(* IEC 61131-3 sources: Lasal/CPU_5344_V01/Class/cmMotor, 1 file *)

(* ---- cmMotor.st ---- *)
(*!
<Class
	Name               = "cmMotor"
	Revision           = "1.0"
	RealtimeTask       = "false"
	CyclicTask         = "true"
	DefCyclictime      = "10 ms"
	BackgroundTask     = "true"
	DefBackground      = "500 ms"
	Sigmatek           = "false"
	OSInterface        = "false"
	HighPriority       = "false"
	Automatic          = "false"
	UpdateMode         = "Prescan"
	SharedCommandTable = "true"
	Objectsize         = "(630,840)">
	<Channels>
		<Server Name="parMinTimeBetweenRev" Visualized="true" Initialize="false" WriteProtected="false" Retentive="File"/>
		<Server Name="parSpeed" Visualized="true" Initialize="false" WriteProtected="false" Retentive="false"/>
		<Server Name="parStartingTime" Visualized="true" Initialize="true" DefValue="2000" WriteProtected="false" Retentive="File"/>
		<Server Name="parTimeOutTime" Visualized="true" Initialize="true" DefValue="20000" WriteProtected="false" Retentive="File"/>
		<Server Name="stsBwd" Visualized="false" Initialize="false" WriteProtected="true" Retentive="false"/>
		<Server Name="stsFwd" Visualized="false" Initialize="false" WriteProtected="true" Retentive="false"/>
		<Server Name="stsStateRun" Visualized="true" Initialize="false" WriteProtected="false" Retentive="false"/>
		<Client Name="iFeedback" Required="false" Internal="false"/>
		<Client Name="iHWAlarm" Required="false" Internal="false" Comment="if used as btb, set sInvert"/>
		<Client Name="iThermFailure" Required="false" Internal="false" Comment="if used, connect thermical failure input,&#13;&#10;normally this input is high if there is a failure&#13;&#10;Else just set sInvert param"/>
		<Client Name="oBwd" Required="false" Internal="false"/>
		<Client Name="oFwd" Required="false" Internal="false"/>
		<Client Name="oSpeed" Required="false" Internal="false"/>
		<Client Name="sInvertFeedback" Required="false" Internal="false"/>
		<Client Name="sInvertHWAlarm" Required="false" Internal="false"/>
		<Client Name="sInvertThermFailure" Required="false" Internal="false"/>
		<Client Name="sMaxSpeedIn" Required="false" Internal="false" DefValue="1000"/>
		<Client Name="sMaxSpeedOut" Required="false" Internal="false" DefValue="10000"/>
		<Client Name="sMinSpeedIn" Required="false" Internal="false" DefValue="0"/>
		<Client Name="sMinSpeedOut" Required="false" Internal="false" DefValue="0"/>
	</Channels>
	<RevDoku>
		<Owner/>
		<Dokumentation Revision="0.1" Date="2019-12-13" Author="JdK&#13;&#10;" Company="vd" Description="calculation speed out is corrected, also added alarm for speed in out of borders"/>
	</RevDoku>
	<Network Name="cmMotor">
		<!-- List of Components in this network -->
		<Components>
			<Object
				Name       = "_base"
				Class      = "cmBase"
				Position   = "(218,120)"
				Visualized = "true">
				<Channels>
					<Server Name="ClassSvr"/>
					<Server Name="cmdHMI"/>
					<Server Name="ErrorNr"/>
					<Server Name="mode"/>
					<Server Name="state"/>
					<Server Name="stsHMI_RunsAllowed"/>
					<Server Name="stsInAlarm"/>
					<Server Name="stsIsInterlocked"/>
					<Client Name="id"/>
					<Client Name="nwEmOrUnit"/>
				</Channels>
			</Object>
		</Components>
		<Comments>
		</Comments>
		<!-- List of Connections in this network -->
		<Connections>
			<Connection Source="this.ClassSvr" Destination="_base.ClassSvr" Vertices="(1036,210),(864,210),"/>
			<Connection Source="this.state" Destination="_base.state" Vertices="(1036,270),(864,270),"/>
			<Connection Source="this.mode" Destination="_base.mode" Vertices="(1036,330),(864,330),"/>
			<Connection Source="this.cmdHMI" Destination="_base.cmdHMI" Vertices="(1036,390),(864,390),"/>
			<Connection Source="this.stsInAlarm" Destination="_base.stsInAlarm" Vertices="(1036,450),(864,510),"/>
			<Connection Source="this.stsIsInterlocked" Destination="_base.stsIsInterlocked" Vertices="(1036,510),(864,570),"/>
			<Connection Source="this.ErrorNr" Destination="_base.ErrorNr" Vertices="(1036,630),(864,690),"/>
			<Connection Source="_base.nwEmOrUnit" Destination="this.nwEmOrUnit" Vertices="(218,210),(38,210),"/>
			<Connection Source="_base.id" Destination="this.id" Vertices="(218,270),(38,270),"/>
			<Connection Source="this.stsHMI_RunsAllowed" Destination="_base.stsHMI_RunsAllowed" Vertices="(1036,570),(864,630),"/>
		</Connections>
		<!-- Headerfiles -->
		<Options>
		</Options>
	</Network>
</Class>
*)
#pragma using cmBase

cmMotor : CLASS
: cmBase
  //Servers:
	stsStateRun 	: SvrCh_motorPos;
	parTimeOutTime 	: SvrCh_UDINT;
	parStartingTime 	: SvrCh_UDINT;
	parMinTimeBetweenRev 	: SvrCh_UDINT;
	parSpeed 	: SvrCh_DINT;
	stsFwd 	: SvrCh_DINT;
	stsBwd 	: SvrCh_DINT;
  //Clients:
	iThermFailure 	: CltCh_DINT;
	iHWAlarm 	: CltCh_DINT;
	iFeedback 	: CltCh_DINT;
	oFwd 	: CltCh_DINT;
	oBwd 	: CltCh_DINT;
	oSpeed 	: CltCh_DINT;
	sInvertThermFailure 	: CltCh_DINT;
	sInvertHWAlarm 	: CltCh_DINT;
	sInvertFeedback 	: CltCh_DINT;
	sMinSpeedOut 	: CltCh_DINT;
	sMaxSpeedOut 	: CltCh_DINT;
	sMinSpeedIn 	: CltCh_DINT;
	sMaxSpeedIn 	: CltCh_DINT;
  //Variables:
		timerFeedback 	: strTimer;
		timerStarting 	: strTimer;
		timerFwdStopped 	: strTimer;
		timerBwdStopped 	: strTimer;
		feedbackConnected 	: DINT;
		tmpOSpeed 	: REAL;
		tmpThermFailure 	: DINT;
		tmpHWAlarm 	: DINT;
		tmpFeedback 	: DINT;
		tmpStartedHMI 	: DINT;
		tmpStartedCS 	: DINT;
		tmpOldSpeed 	: DINT;
  //Functions:

	FUNCTION VIRTUAL GLOBAL Background
		VAR_INPUT
			EAX 	: UDINT;
		END_VAR
		VAR_OUTPUT
			state (EAX) 	: UDINT;
		END_VAR;

	FUNCTION VIRTUAL execHmiCmd1;

	FUNCTION VIRTUAL execHmiCmd2;

	FUNCTION VIRTUAL interlock;

	FUNCTION VIRTUAL work;

	FUNCTION VIRTUAL execStop;

	FUNCTION VIRTUAL Init1;

	FUNCTION VIRTUAL preScanOverride;

	FUNCTION VIRTUAL postScanOverride;

	FUNCTION GLOBAL csStartFwd
		VAR_INPUT
			speed 	: DINT;
		END_VAR;

	FUNCTION GLOBAL csStartBwd
		VAR_INPUT
			speed 	: DINT;
		END_VAR;

	FUNCTION GLOBAL csStop;

	FUNCTION StartFwd;

	FUNCTION StartBwd;

	FUNCTION StopRunning;

	FUNCTION GLOBAL updateSpeed
		VAR_INPUT
			speed 	: DINT;
		END_VAR;
  //Tables:
	FUNCTION @STD
		VAR_OUTPUT
			ret_code	: CONFSTATES;
		END_VAR;
	FUNCTION GLOBAL TAB @CT_;
END_CLASS;

// JdK 13-12-2019 updated calculation of speed, added alarm for speed in out of borders
// JdK 17-5-2019 class motor, created for library icm project 4284 TraffiRoad
// goal is to control motor
// Alarm errornrs:
//                  1: thermicall failure
//                  2: controller failure
//                  3: time-out feedback
//                  4: feedback gone during running
//                  5: speed in out of borders

// HMI cmd1: start run FWD, cmd2: start run Bwd, stop: stop running

FUNCTION VIRTUAL cmMotor::execHmiCmd1

  //start running FWD
  tmpOldSpeed:= parSpeed;
  StartFwd();
  tmpStartedHMI:=1; //rembember who started the motor
  tmpStartedCS:=0;

END_FUNCTION

FUNCTION VIRTUAL cmMotor::execHmiCmd2

  //start running REV
  tmpOldSpeed:= parSpeed;
  StartBwd();
  tmpStartedHMI:=1;//remember who started this
  tmpStartedCS:=0;

END_FUNCTION

FUNCTION GLOBAL cmMotor::csStartFwd
	VAR_INPUT
		speed 	: DINT;
	END_VAR

  //start command from above, only if in auto or service
  IF pmlCom.sts.mode= auto | pmlCom.sts.mode= service THEN
    tmpOldSpeed:= parSpeed;
    parSpeed:=speed;
    StartFwd();
  END_IF;
  tmpStartedHMI:=0; //rembember who started the motor
  tmpStartedCS:=1;

END_FUNCTION

FUNCTION GLOBAL cmMotor::csStartBwd
	VAR_INPUT
		speed 	: DINT;
	END_VAR

  //start command from above, only if in auto or service
  IF pmlCom.sts.mode= auto | pmlCom.sts.mode= service THEN
    tmpOldSpeed:= parSpeed;
    parSpeed:=speed;
    StartBwd();
  END_IF;
  tmpStartedHMI:=0; //rembember who started the motor
  tmpStartedCS:=1;

END_FUNCTION

FUNCTION GLOBAL cmMotor::csStop

  //start command from above, only if in auto or service, or during resetting
  IF pmlCom.sts.mode= auto | pmlCom.sts.mode= service THEN
    StopRunning();
  END_IF;

END_FUNCTION

FUNCTION cmMotor::StartFwd

  IF stsStateRun = moOff | (stsBwd = 1) THEN //only allowed to start if
    stsFwd:=1;
    stsBwd:=0;
    stsStateRun:= moChangeDir;
  ELSIF parSpeed<> tmpOldSpeed & feedbackConnected THEN //JdK 22-4-2022, if speed is changing and feedback is used, change to wait for feedback again
    stsStateRun:= moWaitFeedback;
  END_IF;
  updateSpeed(speed:=parSpeed);

END_FUNCTION

FUNCTION cmMotor::StartBwd

  IF stsStateRun = moOff | (stsBwd = 1) THEN //only allowed to start if
    stsFwd:=0;
    stsBwd:=1;
    stsStateRun:= moChangeDir;
  ELSIF parSpeed<> tmpOldSpeed & feedbackConnected THEN //JdK 22-4-2022, if speed is changing and feedback is used, change to wait for feedback again
    stsStateRun:= moWaitFeedback;
  END_IF;
  updateSpeed(speed:=parSpeed);

END_FUNCTION

FUNCTION cmMotor::StopRunning

  stsStateRun:= moOff;

END_FUNCTION

FUNCTION GLOBAL cmMotor::updateSpeed
	VAR_INPUT
		speed 	: DINT;
	END_VAR

  parSpeed:=speed;
  IF parSpeed > sMaxSpeedIn | parSpeed < sMinSpeedIn THEN
    giveAlarm(errorNr:=5);
  ELSIF sMaxSpeedIn-sMinSpeedIn<>0 THEN
    tmpOSpeed:=((to_real(parSpeed-sMinSpeedIn)/to_real(sMaxSpeedIn-sMinSpeedIn)))*to_real(sMaxSpeedOut-sMinSpeedOut)+to_real(sMinSpeedOut);
    oSpeed:=to_dint(tmpOSpeed);
  ELSE
    oSpeed:=0;
  END_IF;
  oSpeed.Write(input:=oSpeed);

END_FUNCTION

FUNCTION VIRTUAL cmMotor::work

  IF pmlCom.sts.isInterlocked & stsStateRun<>moOff THEN //at interlock, always stop motor
    stsStateRun:=moOff;
  END_IF;

  CASE stsStateRun OF

    moOff: //just do nothing,

    moChangeDir: //wait until change direction is allowed
      IF (timerFwdStopped.done=1 | stsFwd=1) & (timerBwdStopped.done=1 | stsBwd=1) THEN
        IF tmpHWAlarm = 0 THEN
          stsStateRun:=moWaitFeedback;
        ELSE
          giveAlarm(errorNr:=2);
          stsStateRun:=moOff;
        END_IF;
      END_IF;

    moWaitFeedback: //wait for feedback, only if not in simu and if feedback is connected
      IF pmlCom.cmd.simulation=allSimu | feedbackConnected=0 | tmpFeedback THEN
        stsStateRun:=moStarting;
      ELSIF timerFeedback.done THEN
        giveAlarm(errorNr:=3);
        stsStateRun:=moOff;
      END_IF;
      oFwd:=stsFwd;
      oBwd:=stsBwd;

    moStarting: //wait certain time, until motor is running fast and stable enough
      IF pmlCom.cmd.simulation<>allSimu & feedbackConnected=1 & tmpFeedback=0 THEN
        giveAlarm(errorNr:=4); //feedback gone during running
        stsStateRun:=moOff;
      ELSIF tmpHWAlarm THEN
        giveAlarm(errorNr:=2); //hardware not ok
        stsStateRun:=moOff;
      ELSIF timerStarting.done THEN
        stsStateRun:=moRunning;
      END_IF;
      oFwd:=stsFwd;
      oBwd:=stsBwd;

    moRunning: //run untill method stop is called
      IF pmlCom.cmd.simulation<>allSimu & feedbackConnected=1 & tmpFeedback=0 THEN
        giveAlarm(errorNr:=4); //feedback gone during running
        stsStateRun:=moOff;
      ELSIF tmpHWAlarm THEN
        giveAlarm(errorNr:=2); //hardware not ok
        stsStateRun:=moOff;
      END_IF;
      oFwd:=stsFwd;
      oBwd:=stsBwd;

  END_CASE;

END_FUNCTION

FUNCTION VIRTUAL GLOBAL cmMotor::Background
	VAR_INPUT
		EAX 	: UDINT;
	END_VAR
	VAR_OUTPUT
		state (EAX) 	: UDINT;
	END_VAR

  //read in slow inputs
  sInvertThermFailure := sInvertThermFailure.Read();
  sInvertHWAlarm := sInvertHWAlarm.Read();
  sInvertFeedback := sInvertFeedback.Read();
  sMinSpeedOut := sMinSpeedOut.Read();
  sMaxSpeedOut := sMaxSpeedOut.Read();
  sMinSpeedIn := sMinSpeedIn.Read();
  sMaxSpeedIn := sMaxSpeedIn.Read();

  state:=1;

END_FUNCTION

FUNCTION VIRTUAL cmMotor::interlock

  pmlCom.sts.isInterlocked:=pmlCom.cmd.interlock | tmpThermFailure=1;

END_FUNCTION

FUNCTION VIRTUAL cmMotor::execStop

  //stop running
  StopRunning();

END_FUNCTION

FUNCTION VIRTUAL cmMotor::Init1

  IF initDone = 0 THEN
    feedbackConnected:=IsClientConnected(#iFeedback);
    initDone:=1;
  END_IF;
END_FUNCTION

FUNCTION VIRTUAL cmMotor::preScanOverride
  //first read inputs
  iThermFailure := iThermFailure.Read();
  iHWAlarm := iHWAlarm.Read();
  iFeedback := iFeedback.Read();

  tmpThermFailure:=(iThermFailure=1 & sInvertThermFailure=0) | (iThermFailure=0 & sInvertThermFailure=1);
  tmpHWAlarm:=(iHWAlarm=1 & sInvertHWAlarm=0) | (iHWAlarm=0 & sInvertHWAlarm=1 & pmlCom.cmd.simulation<>allSimu);
  tmpFeedback:=(iFeedback=1 & sInvertFeedback=0) | (iFeedback=0 & sInvertFeedback=1);

  //give alarm if there is a thermical failure
  IF tmpThermFailure THEN
    giveAlarm(errorNr:=1);
  END_IF;

  //run timers
  timerFeedback:=runTimer(Active:=stsStateRun=moWaitFeedback, iMem:=timerFeedback, TimerTime:=parTimeOutTime, Pause:=0);
  timerFwdStopped:=runTimer(Active:=oFwd=0, iMem:=timerFwdStopped, TimerTime:=parMinTimeBetweenRev, Pause:=0);
  timerBwdStopped:=runTimer(Active:=oBwd=0, iMem:=timerBwdStopped, TimerTime:=parMinTimeBetweenRev, Pause:=0);
  timerStarting:=runTimer(Active:=stsStateRun=moStarting, iMem:=timerStarting, TimerTime:=parStartingTime, Pause:=0);

  //set outputs to 0
  oFwd:=0;
  oBwd:=0;

  IF tmpStartedHMI=1 & pmlCom.sts.mode<> manual & pmlCom.sts.mode<> service & stsStateRun<>moOff THEN //started in manual, not manual anymore and still running
    StopRunning(); //stop it
  ELSIF tmpStartedCS=1 & pmlCom.sts.mode<> halfAuto & pmlCom.sts.mode<> auto & pmlCom.sts.mode<> service & stsStateRun<> moOff THEN //started from above in auto/half auto, and not in same mode and still running
    StopRunning(); //stop it
  END_IF;

END_FUNCTION

FUNCTION VIRTUAL cmMotor::postScanOverride

  oFwd.Write(input:=oFwd);
  oBwd.Write(input:=oBwd);

END_FUNCTION
